// ---- Trash/MainScreen_1.TcVIS
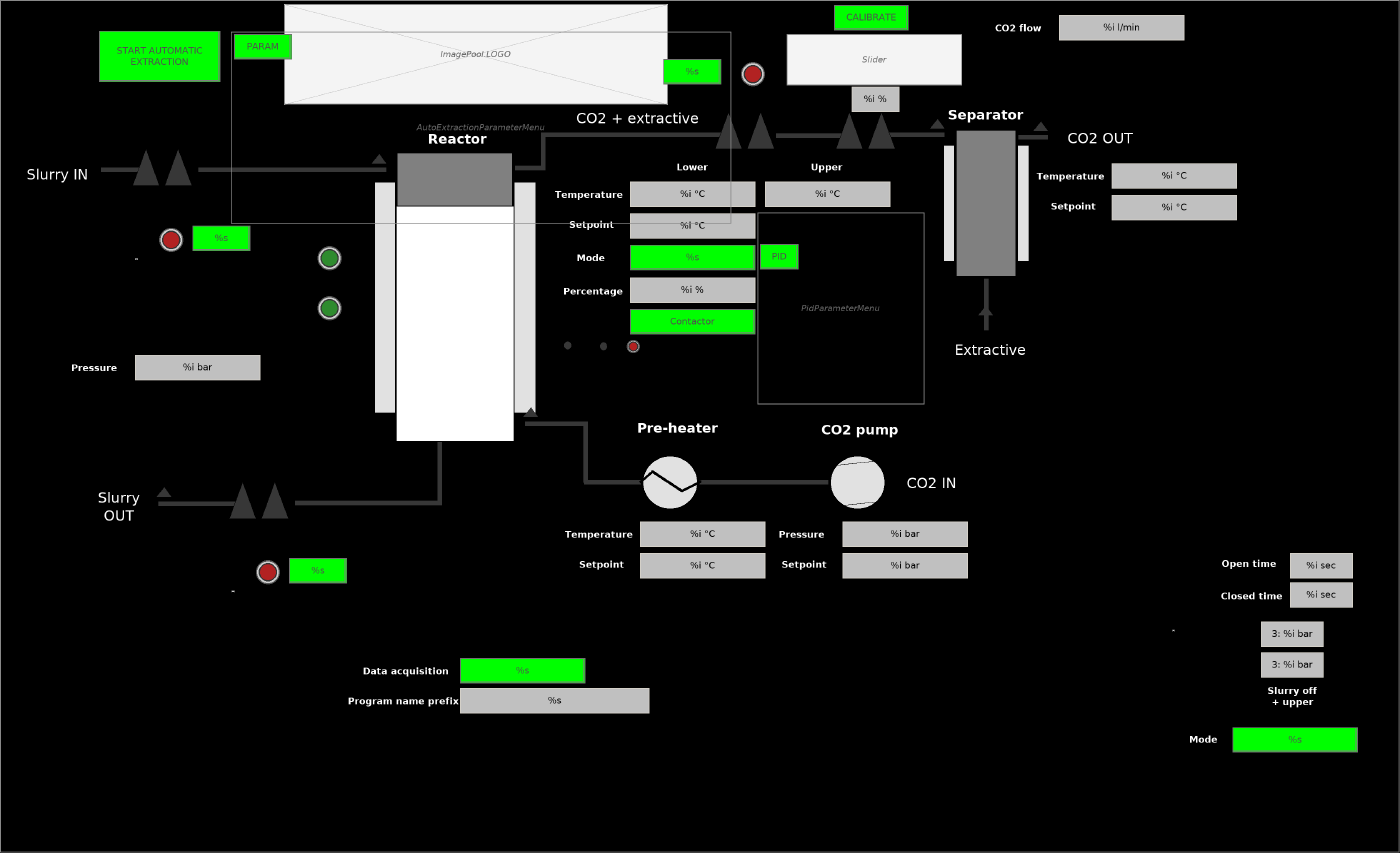
VISUALIZATION MainScreen_1  // 1680x1024
    Line (473,367) (407,367)
    Line (473,308) (407,308)
    Rectangle (1181,326 5x70)
    Rectangle (701,576 350x5)
    Rectangle (525,526 5x80), colour toggle: MainScreenBindings.SlurryOutLine1_ToggleColor
    Rectangle (190,602 100x5), colour toggle: MainScreenBindings.SlurryOutLine1_ToggleColor
    Rectangle (354,601 175x5), colour toggle: MainScreenBindings.SlurryOutLine1_ToggleColor
    Rectangle (121,201 50x5), colour toggle: MainScreenBindings.SlurryInArrow_ToggleColor
    Polygon (446,196) (455,185) (463,196) (457,196) (452,196), colour toggle: MainScreenBindings.SlurryInArrow_ToggleColor
    Rectangle (238,201 225x5), colour toggle: MainScreenBindings.SlurryInArrow_ToggleColor
    Textfield (918,218 150x30), "%i °C", text variable: MainScreenBindings.ReactorUpperTemperatureTextField_TextVariable
    Rectangle (1130,172 107x144)
    Rectangle (447,216 198x282), colour toggle: MainScreenBindings.ReactorBackgroundRectangle_ToggleColor
    RoundedRectangle (474,181 143x345)
    Button (756,371 150x30), "Contactor", colour toggle: MainScreenBindings.ReactorTemperatureContactorLamp_Variable, invisible if: MainScreenBindings.ReactorTemperatureContactorButton_Invisible
        toggle MainScreenBindings.ReactorTemperatureContactorButton_ToggleVariable p2164770859=TRUE
    Lamp1 (746,407 28x18), variable: MainScreenBindings.ReactorTemperatureContactorLamp_Variable, style: Lamp-Lamp1-Red
    Lamp1 (379,351 33x38), variable: MainScreenBindings.ReactorLowerLevelLamp, style: Lamp-Lamp1-Green
    Lamp1 (379,291 33x38), variable: MainScreenBindings.ReactorUpperLevelLamp_Variable, style: Lamp-Lamp1-Green
    Textfield (756,256 150x30), "%i °C", text variable: MainScreenBindings.ReactorTemperatureSetpointTextField_TextVariable
        OnMouseDown: write the text variable via VisuDialogs.Numpad, min 40, max 120
    Label (636,212 142x44), "Temperature"
    Button (756,294 150x30), "%s", text variable: MainScreenBindings.RectorTemperatureControlModeButton_TextVariable, colour toggle: MainScreenBindings.PidParamMenuButton_Invisible
        toggle MainScreenBindings.RectorTemperatureControlModeButton_ToggleVariable
    Label (638,288 142x44), "Mode"
    Label (639,248 142x44), "Setpoint"
    Textfield (756,218 150x30), "%i °C", text variable: MainScreenBindings.ReactorLowerTemperatureTextField_TextVariable
    Label (474,152 150x30), "Reactor"
    RoundedRectangle (474,367 143x162), invisible if: MainScreenBindings.ReactorLowerLevelReactangle_Invisible
    RoundedRectangle (474,307 143x223), invisible if: MainScreenBindings.ReactorUpperLevelRectangle_Invisible
    RoundedRectangle (475,247 142x283), invisible if: MainScreenBindings.ReactorUpperUpperLevelReactangle_Invisible
    Image (278,709 3x1), image: VisuSymbols.Symbols.TriangleRight
    Line (354,638) (288,638)
    Lamp1 (305,668 33x38), variable: MainScreenBindings.SlurryOutValveLamp_Variable, style: Lamp-Lamp1-Red
    Label (641,328 142x44), "Percentage", invisible if: MainScreenBindings.PercentageLabel_Invisible
    Textfield (756,333 150x30), "%i %", text variable: MainScreenBindings.ReactorTemperatureControlPercentageTextField_TextVariable, invisible if: MainScreenBindings.ReactorTemperatureControlPercentageTextField_Invisible
        OnMouseDown: write the text variable via VisuDialogs.Numpad, min 0, max 100
    Label (1373,866 142x44), "Mode", invisible if: true
    Button (1479,873 150x30), "%s", text variable: MainScreenBindings.SlurryOutControlModeButton_TextVariable, colour toggle: MainScreenBindings.SlurryOutControlModeButton_ToggleColor, invisible if: true
        toggle MainScreenBindings.SlurryOutControlModeButton_ToggleVariable
    Button (347,670 69x30), "%s", text variable: MainScreenBindings.SlurryOutValveButton_TextVariable, colour toggle: MainScreenBindings.SlurryOutValveButton_ToggleColor, invisible if: MainScreenBindings.SlurryOutValveButton_Invisible
        toggle MainScreenBindings.SlurryOutValveButton_ToggleVariable
    Image (341,5 460x120), image: ImagePool.LOGO
    Button (912,293 46x30), "PID", invisible if: MainScreenBindings.PidParamMenuButton_Invisible
        toggle MainScreenBindings.PidParamMenuButton_ToggleVariable
    Frame (909,255 200x230), invisible if: MainScreenBindings.PidParamMenuFrame_Invisible
        shows PidParameterMenu()
    Label (42,420 142x44), "Pressure"
    Textfield (162,426 150x30), "%i bar", text variable: MainScreenBindings.ReactorPressureTextField_TextVariable
    Button (552,790 150x30), "%s", text variable: MainScreenBindings.StartMatlabButton_TextVariable, pressed state: RunMATLAB.bMatlabBtnState, input disabled if: MainScreenBindings.StartMatlabButton_DeactivateInputs
        p2175578022: MainScreenBindings.StartMatlabButton_Color
        toggle MainScreenBindings.StartMatlabButton_ToggleVariable
    Image (162,310 3x1), image: VisuSymbols.Symbols.TriangleRight
    Line (238,239) (172,239)
    Lamp1 (189,269 33x38), variable: MainScreenBindings.SlurryInValveLamp_Variable, style: Lamp-Lamp1-Red
    Button (231,271 69x30), "%s", text variable: MainScreenBindings.SlurryInValveControlModeButton_TextVariable, colour toggle: MainScreenBindings.SlurryInValveControlModeButton_ToggleColor, invisible if: MainScreenBindings.SlurryInValveControlModeButton_Invisible
        toggle MainScreenBindings.SlurryInValveControlModeButton_ToggleVariable
    Image (1407,756 2x1), image: VisuSymbols.Symbols.ArrowBoldRight
    Ellipse (769,545 70x68)
    Polyline (768,579) (783,566) (818,589) (840,578) (838,578)
    Ellipse (994,545 70x68)
    Line (994,559) (1052,553)
    Line (994,608) (1052,602)
    Label (648,620 142x44), "Temperature"
    Textfield (768,664 150x30), "%i °C", text variable: MainScreenBindings.PreHeaterTemperatureSetpointTextField_TextVariable
        OnMouseDown: write MainScreenBindings.PreHeaterTemperatureSetpointTextField_WriteAvariable via VisuDialogs.Numpad, min 0, max 120
    Label (651,656 142x44), "Setpoint"
    Textfield (768,626 150x30), "%i °C", text variable: MainScreenBindings.PreHeaterTemperatureTextField_TextVariable
    Label (891,620 142x44), "Pressure"
    Textfield (1011,664 150x30), "%i bar", text variable: MainScreenBindings.Co2PressureSetpointTextField_TextVariable
        OnMouseDown: write MainScreenBindings.Co2PressureSetpointTextField_WriteAvariable via VisuDialogs.Numpad, min 80, max 350
    Label (894,656 142x44), "Setpoint"
    Textfield (1011,626 150x30), "%i bar", text variable: MainScreenBindings.Co2PressureTextField_TextVariable
    Label (1073,565 90x30), "CO2 IN"
    Label (957,501 150x30), "CO2 pump"
    Label (738,499 150x30), "Pre-heater"
    Label (98,574 90x69), "Slurry OUT"
    Label (24,175 90x69), "Slurry IN"
    Label (1151,12 142x44), "CO2 flow"
    Textfield (1271,18 150x30), "%i l/min", text variable: MainScreenBindings.Co2FlowTextField_TextVariable
    RoundedRectangle (1145,154 76x180)
    Label (1108,123 150x30), "Separator"
    Label (654,127 222x30), "CO2 + extractive"
    Label (1254,151 133x30), "CO2 OUT"
    Label (1122,405 133x30), "Extractive"
    Label (1214,190 142x44), "Temperature"
    Textfield (1334,234 150x30), "%i °C", text variable: MainScreenBindings.SeparatorTemperatureSetpointTextField_TextVariable
        OnMouseDown: write MainScreenBindings.SeparatorTemperatureSetpointTextField_WriteAvariable via VisuDialogs.Numpad, min 0, max 100
    Label (1217,226 142x44), "Setpoint"
    Textfield (1334,196 150x30), "%i °C", text variable: MainScreenBindings.SeperatorTemperatureTextField_TextVariable
    Label (416,784 142x44), "Data acquisition"
    Label (1451,655 100x44), "Open time", invisible if: true
    Label (1452,694 100x44), "Closed time", invisible if: true
    Textfield (1548,664 75x30), "%i sec", text variable: MainScreenBindings.SlurryInValveOpenTimeTextField_TextVariable, invisible if: true
        OnMouseDown: write the text variable via VisuDialogs.Numpad, min 0, max 100
    Textfield (1548,699 75x30), "%i sec", text variable: MainScreenBindings.SlurryInValveClosedTimeTextField_TextVariable, invisible if: true
        OnMouseDown: write the text variable via VisuDialogs.Numpad, min 0, max 200
    Label (760,179 142x44), "Lower"
    Label (921,179 142x44), "Upper"
    Textfield (1513,746 75x30), "3: %i bar", text variable: MainScreenBindings.UpperIntervalSlurryOffUpperTextField_TextVariable, invisible if: true
        OnMouseDown: write the text variable via VisuDialogs.Numpad, min -100, max 100
    Textfield (1513,783 75x30), "3: %i bar", text variable: MainScreenBindings.LowerIntervalSlurryOffUpperTextField_TextVariable, invisible if: true
        OnMouseDown: write the text variable via VisuDialogs.Numpad, min -100, max 100
    Label (1515,814 72x44), "Slurry off + upper", invisible if: true
    Textfield (552,826 227x30), "%s", text variable: MainScreenBindings.ProgramNamePrefixTextField_TextVariable
        OnMouseDown: write the text variable via Edit
    Label (413,820 142x44), "Program name prefix"
    Line (677,415) (644,415)
    Ellipse (676,409 10x11)
    Line (719,415) (686,415), invisible if: MainScreenBindings.ReactorTemperatureContactorClosedLine_Invisible
    Ellipse (719,410 10x11)
    Line (725,400) (692,400), invisible if: MainScreenBindings.ReactorTemperatureContactorOpenLine_Invisible
    Line (746,415) (728,415)
    Frame (168,183 71x44)
        shows Valve(valve_toggleColor := MainScreenBindings.SlurryInValveFrame_valve_toggleColor, valve_tapVariable := MainScreenBindings.SlurryInValveFrame_valve_tapVariable)
    Frame (284,583 71x44)
        shows Valve(valve_toggleColor := MainScreenBindings.SlurryOutValveFrame_valve_toggleColor, valve_tapVariable := MainScreenBindings.SlurryOutValveFrame_valve_tapVariable)
    Polygon (188,596) (197,585) (205,596) (199,596) (194,596), colour toggle: MainScreenBindings.SlurryOutLine1_ToggleColor
    Polygon (628,500) (637,489) (645,500) (639,500) (634,500)
    Rectangle (630,506 75x5)
    Rectangle (700,507 5x72)
    Rectangle (650,159 230x5), colour toggle: MainScreenBindings.ExtractiveOutLines_ToggleColor
    Polygon (1116,154) (1125,143) (1133,154) (1127,154) (1122,154), colour toggle: MainScreenBindings.ExtractiveOutLines_ToggleColor
    Rectangle (649,159 5x45), colour toggle: MainScreenBindings.ExtractiveOutLines_ToggleColor
    Rectangle (618,199 35x5), colour toggle: MainScreenBindings.ExtractiveOutLines_ToggleColor
    Polygon (1174,378) (1183,367) (1191,378) (1185,378) (1180,378)
    Rectangle (1222,162 35x5)
    Polygon (1240,157) (1249,146) (1257,157) (1251,157) (1246,157)
    Line (936,127) (870,127)
    Lamp1 (887,70 33x38), variable: MainScreenBindings.ExtractiveOutOnOffValveLamp_variable, style: Lamp-Lamp1-Red
    Rectangle (931,160 90x5), colour toggle: MainScreenBindings.ExtractiveOutLines_ToggleColor
    Frame (867,139 71x44)
        shows Valve(valve_toggleColor := MainScreenBindings.ExtractiveOutletOnOff_Valve_ToggleColor, valve_tapVariable := MainScreenBindings.ExtractiveOutletOnOff_Valve_TapVariable)
    Button (796,71 69x30), "%s", text variable: MainScreenBindings.ExtractiveOutOnOffValveButton_TextVariable, colour toggle: MainScreenBindings.ExtractiveOutOnOffValveButton_ToggleColor
        toggle MainScreenBindings.ExtractiveOutOnOffValveButton_ToggleVariable
    Line (1065,129) (1016,129)
    Rectangle (1063,159 70x5), colour toggle: MainScreenBindings.ExtractiveOutLines_ToggleColor
    Frame (1012,139 71x44)
        shows Valve(valve_toggleColor := MainScreenBindings.ExtractiveOutletOnOff_Valve_ToggleColor, valve_tapVariable := MainScreenBindings.ExtractiveOutletOnOff_Valve_TapVariable)
    Button (1001,6 89x30), "CALIBRATE", invisible if: MainScreenBindings.ExtractiveOutletValveSlider_DisableInputs
        tap MainScreenBindings.ExtractiveOutletValveCalibrateButton_TapVariable
    Slider (944,41 210x61), variable: MainScreenBindings.ExtractiveOutletValveSlider_Variable, invisible if: MainScreenBindings.ExtractiveOutletValveSlider_Invisible, input disabled if: MainScreenBindings.ExtractiveOutletValveSlider_DisableInputs, scale 0..10
    Button (119,37 145x61), "START AUTOMATIC EXTRACTION", text variable: MainScreenBindings.ExtractiveOutOnOffValveButton_TextVariable, colour toggle: MainScreenBindings.StartAutomaticExtractionButton_ToggleVariable, input disabled if: MainScreenBindings.StartAutomaticExtractionButton_DeactivateInputs
        toggle MainScreenBindings.StartAutomaticExtractionButton_ToggleVariable
    Button (281,41 69x30), "PARAM", text variable: MainScreenBindings.SlurryInValveControlModeButton_TextVariable
        toggle MainScreenBindings.autoExtractionParameterMenuButton_ToggleVariable
    Frame (277,38 600x230), invisible if: MainScreenBindings.autoExtractionParameterMenuFrame_Invisible
        shows AutoExtractionParameterMenu()
    Textfield (1022,104 57x30), "%i %", text variable: MainScreenBindings.ControlValveOpeningPercentageTextBox_TextVariable
END_VISUALIZATION

// ---- Trash/MainScreen_OLD.TcVIS
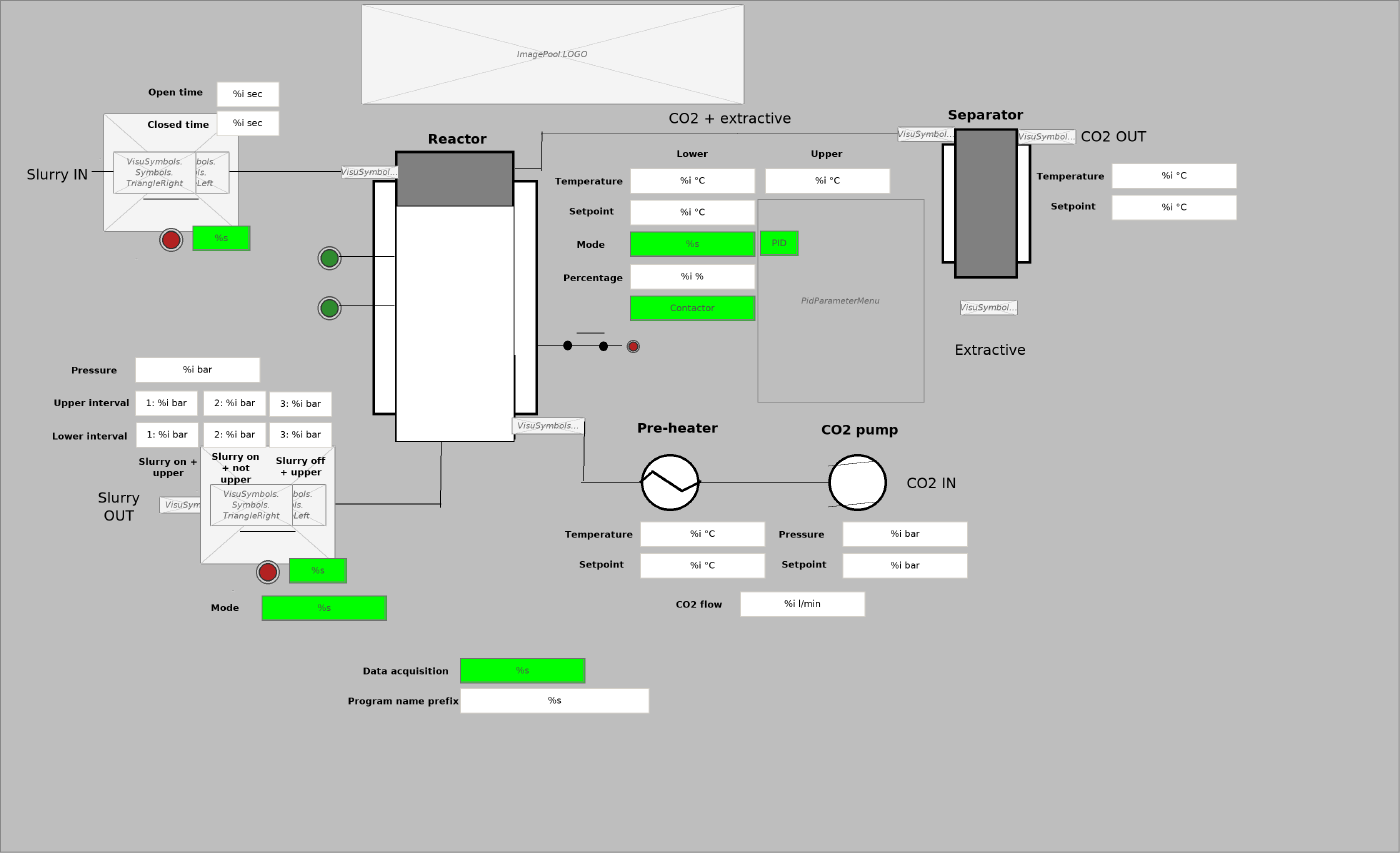
VISUALIZATION MainScreen_OLD  // 1680x1024
    Textfield (918,202 150x30), "%i °C", text variable: ReactorTemperatureControl.iTemperatureLowerDisplayValue
    Rectangle (1130,172 107x144)
    Image (124,136 162x142), invisible if: NOT GVL_IO.reactorInletValve, image: ImagePool.VALVE
    Rectangle (447,216 198x282), colour toggle: (ReactorTemperatureControl.bTemperatureControlSwitch) OR (ReactorTemperatureControl.iTemperatureControlPercentage > 0) OR ((ReactorTemperatureControl.iTemperatureControlPercentage = 0) AND (GVL_IO.reactorTemperatureContactor = 1))
    RoundedRectangle (474,181 143x345)
    Button (756,355 150x30), "Contactor", colour toggle: GVL_IO.reactorTemperatureContactor, invisible if: ReactorTemperatureControl.iTemperatureControlPercentage > 0 or ReactorTemperatureControl.bTemperatureControlSwitch= 1
        toggle GVL_IO.reactorTemperatureContactor
    Lamp1 (746,407 28x18), variable: GVL_IO.reactorTemperatureContactor, style: Lamp-Lamp1-Red
    Lamp1 (379,351 33x38), variable: GVL_IO.reactorLevelLow, style: Lamp-Lamp1-Green
    Lamp1 (379,291 33x38), variable: GVL_IO.reactorLevelHigh, style: Lamp-Lamp1-Green
    Textfield (756,240 150x30), "%i °C", text variable: ReactorTemperatureControl.iTemperatureSetpoint
        OnMouseDown: write the text variable via VisuDialogs.Numpad, min 40, max 120
    Label (636,196 142x44), "Temperature"
    Button (756,278 150x30), "%s", text variable: ReactorTemperatureControl.sTemperatureControlState, colour toggle: ReactorTemperatureControl.bTemperatureControlSwitch
        toggle ReactorTemperatureControl.bTemperatureControlSwitch
    Label (638,272 142x44), "Mode"
    Label (639,232 142x44), "Setpoint"
    Textfield (756,202 150x30), "%i °C", text variable: ReactorTemperatureControl.iTemperatureDisplayValue
    Line (529,526) (528,609)
    Line (529,605) (363,605)
    Line (473,367) (407,367)
    Line (473,308) (407,308)
    RoundedRectangle (474,426 144x101), invisible if: (NOT GVL_IO.reactorLevelLowerLow) OR (GVL_IO.reactorLevelHigh)
    Label (474,152 150x30), "Reactor"
    RoundedRectangle (474,367 143x162), invisible if: (NOT GVL_IO.reactorLevelHigh) OR (GVL_IO.reactorLevelLow)
    RoundedRectangle (474,307 143x223), invisible if: (NOT GVL_IO.reactorLevelLow) OR (GVL_IO.reactorLevelHigherHigh)
    RoundedRectangle (475,247 142x283), invisible if: (NOT GVL_IO.reactorLevelHigherHigh)
    Image (191,596 88x20), image: VisuSymbols.Symbols.ArrowBoldLeft
    Image (240,535 162x142), invisible if: NOT GVL_IO.reactorOutletValve, image: ImagePool.VALVE
    Image (292,581 99x50), invisible if: GVL_IO.reactorOutletValve, image: VisuSymbols.Symbols.TriangleLeft
    Image (278,709 3x1), image: VisuSymbols.Symbols.TriangleRight
    Image (252,581 99x50), invisible if: GVL_IO.reactorOutletValve, image: VisuSymbols.Symbols.TriangleRight
    Line (354,638) (288,638)
    Lamp1 (305,668 33x38), variable: GVL_IO.reactorOutletValve, style: Lamp-Lamp1-Red
    Label (641,312 142x44), "Percentage", invisible if: ReactorTemperatureControl.bTemperatureControlSwitch
    Textfield (756,317 150x30), "%i %", text variable: ReactorTemperatureControl.iTemperatureControlPercentage, invisible if: ReactorTemperatureControl.bTemperatureControlSwitch
        OnMouseDown: write the text variable via VisuDialogs.Numpad, min 0, max 100
    Label (199,708 142x44), "Mode"
    Button (314,715 150x30), "%s", text variable: ReactorLevelAndPressureControl.sLevelControlState, colour toggle: ReactorLevelAndPressureControl.bLevelControlSwitch
        toggle ReactorLevelAndPressureControl.bLevelControlSwitch
    Button (347,670 69x30), "%s", text variable: ReactorLevelAndPressureControl.sLevelValveState, colour toggle: GVL_IO.reactorOutletValve, invisible if: ReactorLevelAndPressureControl.sLevelControlState = 'AUTO'
        toggle GVL_IO.reactorOutletValve
    Line (414,206) (248,206)
    Image (235,589 2x1), image: VisuSymbols.Symbols.ArrowBoldRight
    Image (409,199 69x15), image: VisuSymbols.Symbols.ArrowBoldRight
    Image (433,5 460x120), image: ImagePool.LOGO
    Button (912,277 46x30), "PID", invisible if: ReactorTemperatureControl.bTemperatureControlSwitch
        toggle ReactorTemperatureControl.bPIDcontrolParameterMenu
    Frame (909,239 200x244), invisible if: MainScreenBindings.PidParamMenuFrame_Invisible
        shows PidParameterMenu()
    Label (42,423 142x44), "Pressure"
    Textfield (162,429 150x30), "%i bar", text variable: ReactorLevelAndPressureControl.iPressureScaledValue
    Button (552,790 150x30), "%s", text variable: RunMATLAB.sMatlabRunningState, pressed state: RunMATLAB.bMatlabBtnState, input disabled if: RunMATLAB.dMatlabBtnColor = 16#FFFFFF00
        p2175578022: RunMATLAB.dMatlabBtnColor
        toggle RunMATLAB.bMatlabBtn
    Line (162,206) (110,206)
    Image (176,182 99x50), invisible if: GVL_IO.reactorInletValve, image: VisuSymbols.Symbols.TriangleLeft
    Image (162,310 3x1), image: VisuSymbols.Symbols.TriangleRight
    Image (136,182 99x50), invisible if: GVL_IO.reactorInletValve, image: VisuSymbols.Symbols.TriangleRight
    Line (238,239) (172,239)
    Lamp1 (189,269 33x38), variable: GVL_IO.reactorInletValve, style: Lamp-Lamp1-Red
    Button (231,271 69x30), "%s", text variable: ReactorLevelAndPressureControl.sFillingValveState, colour toggle: GVL_IO.reactorInletValve, invisible if: ReactorLevelAndPressureControl.sLevelControlState = 'AUTO'
        toggle GVL_IO.reactorInletValve
    Image (119,190 2x1), image: VisuSymbols.Symbols.ArrowBoldRight
    Image (614,501 88x20), image: VisuSymbols.Symbols.ArrowBoldLeft
    Line (701,506) (700,577)
    Line (1001,579) (697,579)
    Ellipse (769,545 70x68)
    Polyline (768,579) (783,566) (818,589) (840,578) (838,578)
    Ellipse (994,545 70x68)
    Line (994,559) (1052,553)
    Line (994,608) (1052,602)
    Label (648,620 142x44), "Temperature"
    Textfield (768,664 150x30), "%i °C", text variable: SerialCommunicationHandler.preHeaterTemperatureSetpoint
        OnMouseDown: write SerialCommunicationHandler.preHeaterTemperatureSetSetpoint via VisuDialogs.Numpad, min 0, max 120
    Label (651,656 142x44), "Setpoint"
    Textfield (768,626 150x30), "%i °C", text variable: SerialCommunicationHandler.preHeaterTemperatureMeasurement
    Label (891,620 142x44), "Pressure"
    Textfield (1011,664 150x30), "%i bar", text variable: SerialCommunicationHandler.pumpingPressureSetpoint
        OnMouseDown: write SerialCommunicationHandler.pumpingPressureSetSetpoint via VisuDialogs.Numpad, min 80, max 350
    Label (894,656 142x44), "Setpoint"
    Textfield (1011,626 150x30), "%i bar", text variable: SerialCommunicationHandler.pumpingPressureMeasurement
    Label (1073,565 90x30), "CO2 IN"
    Label (957,501 150x30), "CO2 pump"
    Label (738,499 150x30), "Pre-heater"
    Label (98,574 90x69), "Slurry OUT"
    Label (24,175 90x69), "Slurry IN"
    Label (768,704 142x44), "CO2 flow"
    Textfield (888,710 150x30), "%i l/min", text variable: SerialCommunicationHandler.flowMeasurement
    Line (649,202) (618,202)
    Line (650,158) (649,205)
    Line (1121,160) (649,161)
    Image (1077,152 69x18), image: VisuSymbols.Symbols.ArrowBoldRight
    RoundedRectangle (1145,154 76x180)
    Label (1108,123 150x30), "Separator"
    Label (765,127 222x30), "CO2 + extractive"
    Image (1152,360 69x18), angle 90, image: VisuSymbols.Symbols.ArrowBoldRight
    Image (1222,155 69x18), image: VisuSymbols.Symbols.ArrowBoldRight
    Label (1270,149 133x30), "CO2 OUT"
    Label (1122,405 133x30), "Extractive"
    Label (1214,190 142x44), "Temperature"
    Textfield (1334,234 150x30), "%i °C", text variable: SerialCommunicationHandler.separatorTemperatureSetpoint
        OnMouseDown: write SerialCommunicationHandler.separatorTemperatureSetSetpoint via VisuDialogs.Numpad, min 0, max 100
    Label (1217,226 142x44), "Setpoint"
    Textfield (1334,196 150x30), "%i °C", text variable: SerialCommunicationHandler.separatorTemperatureMeasurement
    Label (416,784 142x44), "Data acquisition"
    Label (60,462 100x44), "Upper interval"
    Label (58,502 100x44), "Lower interval"
    Textfield (162,469 75x30), "1: %i bar", text variable: ReactorLevelAndPressureControl.PressureUpperInterVal_1
        OnMouseDown: write the text variable via VisuDialogs.Numpad, min -100, max 100
    Textfield (244,469 75x30), "2: %i bar", text variable: ReactorLevelAndPressureControl.PressureUpperInterVal_2
        OnMouseDown: write the text variable via VisuDialogs.Numpad, min -100, max 100
    Textfield (163,507 75x30), "1: %i bar", text variable: ReactorLevelAndPressureControl.PressureLowerInterval_1
        OnMouseDown: write the text variable via VisuDialogs.Numpad, min -100, max 100
    Textfield (244,507 75x30), "2: %i bar", text variable: ReactorLevelAndPressureControl.PressureLowerInterval_2
        OnMouseDown: write the text variable via VisuDialogs.Numpad, min -100, max 100
    Label (163,89 100x44), "Open time"
    Label (164,128 100x44), "Closed time"
    Textfield (260,98 75x30), "%i sec", text variable: ReactorLevelAndPressureControl.fillingValveOpenInterval
        OnMouseDown: write the text variable via VisuDialogs.Numpad, min 0, max 100
    Textfield (260,133 75x30), "%i sec", text variable: ReactorLevelAndPressureControl.fillingValveCloseInterval
        OnMouseDown: write the text variable via VisuDialogs.Numpad, min 0, max 200
    Label (760,163 142x44), "Lower"
    Label (921,163 142x44), "Upper"
    Textfield (323,470 75x30), "3: %i bar", text variable: ReactorLevelAndPressureControl.PressureUpperInterVal_3
        OnMouseDown: write the text variable via VisuDialogs.Numpad, min -100, max 100
    Textfield (323,507 75x30), "3: %i bar", text variable: ReactorLevelAndPressureControl.PressureLowerInterval_3
        OnMouseDown: write the text variable via VisuDialogs.Numpad, min -100, max 100
    Label (163,539 78x44), "Slurry on + upper"
    Label (325,538 72x44), "Slurry off + upper"
    Label (247,540 72x44), "Slurry on + not upper"
    Textfield (552,826 227x30), "%s", text variable: GVL_OPC.OPC_ProgramNamePrefix
        OnMouseDown: write the text variable via Edit
    Label (413,820 142x44), "Program name prefix"
    Line (677,415) (644,415)
    Ellipse (676,409 10x11)
    Line (719,415) (686,415), invisible if: NOT GVL_IO.reactorTemperatureContactor
    Ellipse (719,410 10x11)
    Line (725,400) (692,400), invisible if: GVL_IO.reactorTemperatureContactor
    Line (746,415) (728,415)
END_VISUALIZATION

// ---- Trash/SerialCommVisuTest.TcVIS
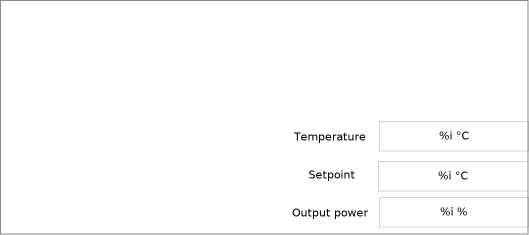
VISUALIZATION SerialCommVisuTest  // 529x235
    Textfield (379,121 150x30), "%i °C", text variable: SerialCommunicationController.pumpingPressureMeasurement
    Label (259,115 142x44), "Temperature"
    Label (259,191 142x44), "Output power"
    Textfield (379,197 150x30), "%i %", text variable: SerialCommunicationController.pumpingPressureOutputPower
    Textfield (378,161 150x30), "%i °C", text variable: SerialCommunicationController.pumpingPressureSetpoint
        OnMouseDown: write SerialCommunicationController.pumpingPressureSetSetpoint via VisuDialogs.Numpad, min 0, max 120
    Label (261,153 142x44), "Setpoint"
END_VISUALIZATION

// ---- Trash/SerialCommVisuTest_1.TcVIS
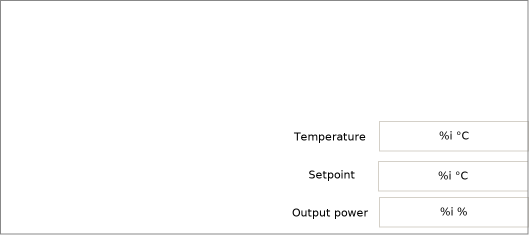
VISUALIZATION SerialCommVisuTest_1  // 529x235
    Textfield (379,121 150x30), "%i °C", text variable: SerialCommunicationController.pumpingPressureMeasurement
    Label (259,115 142x44), "Temperature"
    Label (259,191 142x44), "Output power"
    Textfield (379,197 150x30), "%i %", text variable: SerialCommunicationController.pumpingPressureOutputPower
    Textfield (378,161 150x30), "%i °C", text variable: SerialCommunicationController.pumpingPressureSetpoint
        OnMouseDown: write SerialCommunicationController.pumpingPressureSetSetpoint via VisuDialogs.Numpad, min 0, max 120
    Label (261,153 142x44), "Setpoint"
END_VISUALIZATION
